{attribute 'linkalways'} 
{attribute 'no_explicit_call' := 'This FB is a CLASS and must be accessed using methods or properties'}
{attribute 'enable_dynamic_creation'}
FUNCTION_BLOCK GraphFramework IMPLEMENTS I_GraphFramework
VAR
	_nodeFactory : NodeFactory;
	_datatypes : Datatypes;
	datatypeNodeFactory : DatatypeNodeFactory(_datatypes, _nodeFactory);
END_VAR

METHOD PUBLIC Create : I_Graph
VAR
	pGraph : POINTER TO Graph;
END_VAR
pGraph := __NEW(Graph(NodeFactory := _nodeFactory));
Create := pGraph^;
END_METHOD

PROPERTY PUBLIC Datatypes : I_Datatypes
GET
Datatypes := _datatypes;
END_GET
END_PROPERTY

METHOD PUBLIC Install
VAR_INPUT
	Pack : I_GraphPack;
END_VAR
Pack.RegisterWithDatatypes(Datatypes);
Pack.RegisterWithNodeFactory(NodeFactory);
END_METHOD

PROPERTY PUBLIC NodeFactory : I_NodeFactory
GET
NodeFactory := _nodeFactory;
END_GET
END_PROPERTY

END_FUNCTION_BLOCK

(* stored: Version 1.1.0.1, ProductVersion 3.1.4024.13
   POU GraphFramework: Id {55908e16-d4de-485c-8d69-f119453fe181}, SpecialFunc None
   Method Create: Id {bb10b59b-8876-48c1-a25f-6c91a750d037}
   Property Datatypes: Id {11db57fe-5650-4afc-a04b-0fd8208f9293}
   Get Get: Id {3e243290-827e-405d-b647-e2ae05f0f9b6}
   Method Install: Id {e4dda167-98bc-0854-02d5-43a8f02f58db}
   Property NodeFactory: Id {2a4f3a49-3a80-4475-bdc3-fa7105b5ece9}
   Get Get: Id {e9e37f33-4e35-454d-aa0b-2af694dba608} *)
